% RSLogix 500 project AND_BAK027.RSS, saved by version 8.10.00.18 %
PROJECT "UNTITLED"    % processor: MicroLogix 1200 %

PROGRAM FILES
  LAD 2   7 rungs

DATA FILES
  O0 OUTPUT  4 elements
  I1 INPUT  4 elements
  S2 STATUS  66 elements
  B3 BINARY  1 elements
  T4 TIMER  1 elements
  C5 COUNTER  1 elements
  R6 CONTROL  1 elements
  N7 INTEGER  1 elements
  F8 FLOAT  1 elements

LADDER 2
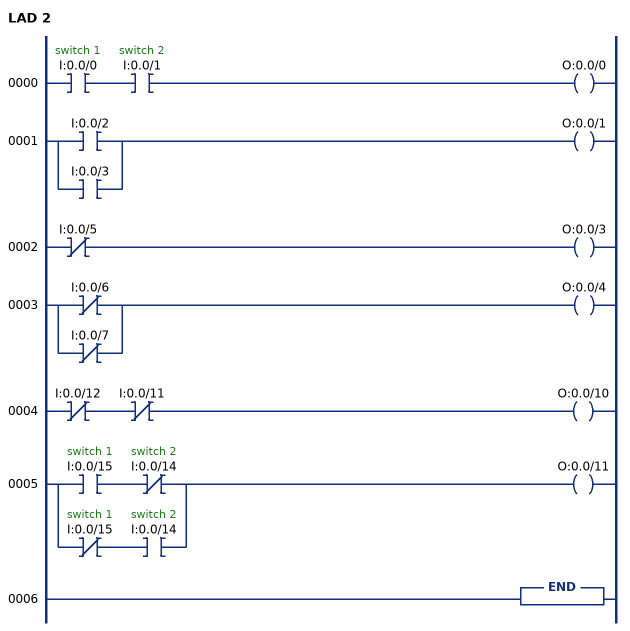
% Rung: 0 %
SOR XIC I:0.0/0 XIC I:0.0/1 OTE O:0.0/0 EOR
%   I:0.0/0  "switch 1" %
%   I:0.0/1  "switch 2" %
% Rung: 1 %
SOR BST XIC I:0.0/2 NXB XIC I:0.0/3 BND OTE O:0.0/1 EOR
% Rung: 2 %
SOR XIO I:0.0/5 OTE O:0.0/3 EOR
% Rung: 3 %
SOR BST XIO I:0.0/6 NXB XIO I:0.0/7 BND OTE O:0.0/4 EOR
% Rung: 4 %
SOR XIO I:0.0/12 XIO I:0.0/11 OTE O:0.0/10 EOR
% Rung: 5 %
SOR BST XIC I:0.0/15 XIO I:0.0/14 NXB XIO I:0.0/15 XIC I:0.0/14 BND OTE O:0.0/11 EOR
%   I:0.0/15  "switch 1" %
%   I:0.0/14  "switch 2" %
% Rung: 6 %
SOR END EOR
